KUKA KRL data list: rs.dat

&ACCESS RVO
&REL 74
DEFDAT rs PUBLIC

GLOBAL STRUC ST_RS BOOL SET, RESET1, Q1
GLOBAL STRUC ST_SR BOOL SET1, RESET, Q1

ENDDAT
